FUNCTION_BLOCK MinutesSinceLastFeedBasic (* Basic Function Block Type *)
  (* Standard: 61499-2 *)
  (* Version 0.0, 7/5/2026, Schneider Electric, Template *)
  PACKAGE SE.Nereda;
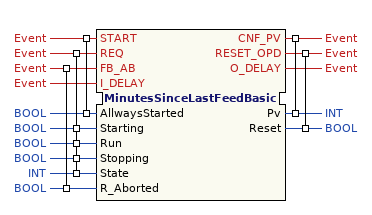
  EVENT_INPUT
    START WITH AllwaysStarted;
    REQ WITH Stopping, Starting, Run, State; (* Normal Execution Request *)
    FB_AB WITH R_Aborted;
    I_DELAY;
  END_EVENT
  EVENT_OUTPUT
    CNF_PV WITH Pv; (* Execution Confirmation *)
    RESET_OPD WITH Reset;
    O_DELAY;
  END_EVENT
  VAR_INPUT
    AllwaysStarted : BOOL;
    Starting : BOOL;
    Run : BOOL;
    Stopping : BOOL;
    State : INT;
    R_Aborted : BOOL;
  END_VAR
  VAR_OUTPUT
    Pv : INT; (* Output event qualifier *)
    Reset : BOOL;
  END_VAR
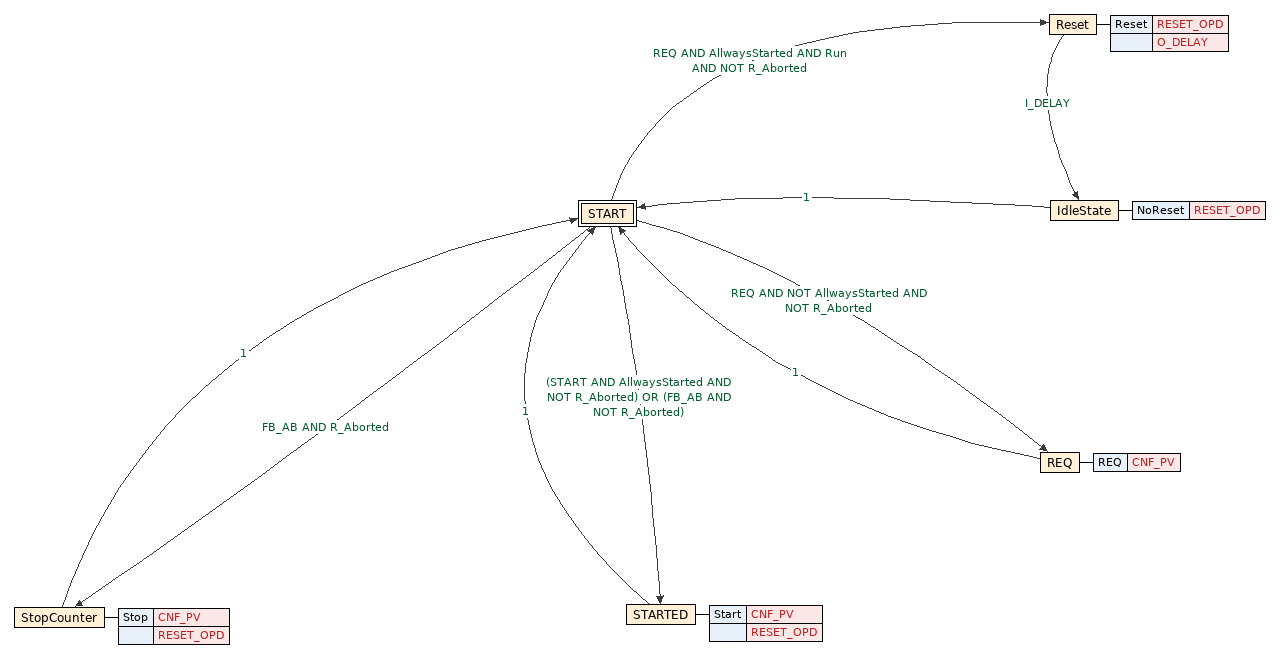
  EC_STATES
    START; (* Initial State *)
    REQ : REQ -> CNF_PV;
    Reset : Reset -> RESET_OPD, -> O_DELAY;
    IdleState : NoReset -> RESET_OPD;
    STARTED : Start -> CNF_PV, -> RESET_OPD;
    StopCounter : Stop -> CNF_PV, -> RESET_OPD;
  END_STATES
  EC_TRANSITIONS
    START TO REQ := REQ AND NOT AllwaysStarted AND NOT R_Aborted;
    REQ TO START := 1;
    START TO Reset := REQ AND AllwaysStarted AND Run AND NOT R_Aborted;
    Reset TO IdleState := I_DELAY;
    START TO STARTED := (START AND AllwaysStarted AND NOT R_Aborted) OR (FB_AB AND NOT R_Aborted);
    STARTED TO START := 1;
    IdleState TO START := 1;
    START TO StopCounter := FB_AB AND R_Aborted;
    StopCounter TO START := 1;
  END_TRANSITIONS
  ALGORITHM REQ IN ST:
;
IF (Starting AND State = 1) OR (Run AND State = 2) OR (Stopping AND State = 3) THEN
	Pv := 1;
ELSE
	Pv := 0;
END_IF;
  END_ALGORITHM
  ALGORITHM Reset IN ST:
;
Reset := TRUE;
  END_ALGORITHM
  ALGORITHM NoReset IN ST:
;
Reset := FALSE;
  END_ALGORITHM
  ALGORITHM Start IN ST:
;
Pv := 1;
Reset := FALSE;
  END_ALGORITHM
  ALGORITHM Stop IN ST:
;
Pv := 0;
Reset := TRUE;
  END_ALGORITHM
END_FUNCTION_BLOCK
